// TIA Portal V17 export
// export: Created 2024-06-14T09:52:56.8973691Z, ExportSetting WithDefaults, DisplayName Totally Integrated Automation Portal, DisplayVersion V17, DisplayName TIA Portal Openness, DisplayVersion V17, DisplayName TIA Portal Version Control Interface, DisplayVersion V17, DisplayName Simotion SCOUT TIA, DisplayVersion 5.4.3.0, DisplayName SINAMICS Startdrive Advanced, DisplayVersion V17 SP1 Update 1, DisplayName SINAMICS Startdrive G110M, G120, G120C, G120D, G120P, G115D, DisplayVersion V17 SP1 Update 1, DisplayName SINAMICS Startdrive G130, G150, S120, S150, SINAMICS MV, S210, DisplayVersion V17 SP1 Update 1, DisplayName STEP 7 Professional, DisplayVersion V17, DisplayName STEP 7 Safety, DisplayVersion V17, DisplayName WinCC Professional, DisplayVersion V17
DATA_BLOCK "fb_Fifo_1_DB_"   // DB51
VERSION : 0.1
// stored: AutoNumber true, DBAccessibleFromOPCUA true, InstanceOfName fb_Fifo, InstanceOfType FB
"fb_Fifo"
   // VAR_INPUT
   //    INxWrite : Bool;
   //    INxRead : Bool;
   // END_VAR
   // VAR_OUTPUT
   //    OUTbStatus : Byte;
   // END_VAR
   // VAR_IN_OUT
   //    IOsFIFO_IN : Array[1..50] of "uCylinderData";
   //    IOsFIFO_OUT : Array[1..50] of "uCylinderData";
   //    IOiIN_Len : Int;
   //    IOiOUT_Len : Int;
   //    IOiNo_Items_Cpy : Int;
   // END_VAR
   // VAR
   //    idx1 { S7_SetPoint := 'True'} : Int;
   //    idx2 { S7_SetPoint := 'True'} : Int;
   //    idx3 { S7_SetPoint := 'True'} : Int;
   //    idx4 : Int;
   //    sEmpty : "uCylinderData";
   // END_VAR
BEGIN
END_DATA_BLOCK
